FUNCTION_BLOCK FB_System_BelAu_Sensorik
VAR_INPUT
END_VAR
VAR_OUTPUT
	(* Dunkelheit Sensor 1*)
	Dunkelheit_OUT	: REAL;
END_VAR
VAR
	(* Hardware oder DALI *)
	Dunkelheit_IN		: REAL;
END_VAR

(* ggfs Umrechung *)
Dunkelheit_OUT := Dunkelheit_IN * 3 ;

END_FUNCTION_BLOCK

(* stored: Version 1.1.0.1, ProductVersion 3.1.4024.9
   POU FB_System_BelAu_Sensorik: Id {83577a62-dd5e-46d6-9e66-a212e4d24a53}, SpecialFunc None *)
